PROGRAM MAIN
VAR
//	stThisIsOurFirstInstanceOfAStructure : ST_Event;
	bBoolean : BOOL;
	eEventType1 : E_EventType := E_EventType.Alarm;
	eEventSeverity1 : TcEventSeverity := TcEventSeverity.Error;
	nEventIdentity1 : UDINT := 42;
	sEventText1 : STRING(255) := 'This is a scarry event';

	CsvPersistentEventStorage : FB_CsvPersistentEventStorage;
	Eventlogger : EventLogger(CsvPersistentEventStorage);
END_VAR

IF bBoolean THEN
	Eventlogger.AddEvent(eEventType1 , eEventSeverity1 , nEventIdentity1 , sEventText1);
	bBoolean := FALSE;
END_IF

CsvPersistentEventStorage();

END_PROGRAM

(* stored: Version 1.1.0.1, ProductVersion 3.1.4024.12
   POU MAIN: Id {43234277-4774-44a3-bd16-428c45b77a36}, SpecialFunc None *)
